{attribute 'qualified_only'}
{attribute 'strict'}
{attribute 'to_string'}
TYPE E_EM_Lift_Seq_ProductionExecute :
(
	Idle := c_nSeqIdle,
	Start := c_nSeqStart,

	
	
	Ready := c_nSeqReady,
	Error := c_nSeqError

);
END_TYPE

(* stored: Version 1.1.0.1, ProductVersion 3.1.4026.13
   DUT E_EM_Lift_Seq_ProductionExecute: Id {9ed95578-29ed-4af7-95b5-3b7ddfb260b1} *)
